Staubli VAL3: editNumField.pgx

public program editNumField(string x_sTitle (dimensions=1), string& x_sItemName[] (dimensions=1), num& x_nItem[] (dimensions=1), num& x_nMin[] (dimensions=1), num& x_nMax[] (dimensions=1))
  local num j
  local num l_nSize
  local num l_nKey
  local string l_sEvent
  local num l_nIndex
  local num l_nField
  local string l_sItem
  local num i
  local string l_sEmpty[2]
  local string l_sString1
  local num l_nFollow
begin
  //  //clear & copy
  //  nView=nFirst=0
  //  call listempty()
  //  call numCopy(x_nItem,nOldValue)
  //  call numCopy(x_nItem,nOffSet)
  //  for j=0 to size(nOffSet)-1
  //    nOffSet[j]=0
  //  endFor
  //  // take the size
  //  l_nSize=size(x_sItemName)-1
  //  // create the LIST
  //  call setSizeList(2,max((6-l_nSize/2)-2,2)-2,20,min((l_nSize+1),12))
  //  call listcreate(x_sTitle)
  //  //
  //  // insert items
  //  //
  //  if nParaAdjustType==1
  //    for j=0 to l_nSize
  //      l_sItem=x_sItemName[j]
  //      if l_sItem!=""
  //        if j==9
  //          call strlength(l_sItem,10)
  //          if x_nItem[j]==0
  //            call listadd(l_sItem+": "+"关")
  //          else
  //            call listadd(l_sItem+": "+"开")
  //          endIf
  //        else
  //          call strlength(l_sItem,10)
  //          call listadd(l_sItem+": "+toString(".3",x_nItem[j]))
  //        endIf
  //        nOffSet[j]=nOffSet[max(j-1,0)]
  //      else
  //        nOffSet[j]=nOffSet[max(j-1,0)]+1
  //      endIf
  //    endFor
  //  endIf
  //  if nParaAdjustType==2
  //    for j=0 to l_nSize
  //      l_sItem=x_sItemName[j]
  //      if l_sItem!=""
  //        if j==7
  //          call strlength(l_sItem,10)
  //          if x_nItem[j]==0
  //            call listadd(l_sItem+": "+"关")
  //          else
  //            call listadd(l_sItem+": "+"开")
  //          endIf
  //        else
  //          call strlength(l_sItem,10)
  //          call listadd(l_sItem+": "+toString(".3",x_nItem[j]))
  //        endIf
  //        nOffSet[j]=nOffSet[max(j-1,0)]
  //      else
  //        nOffSet[j]=nOffSet[max(j-1,0)]+1
  //      endIf
  //    endFor
  //  endIf
  //  if nParaAdjustType==3
  //    for j=0 to l_nSize
  //      l_sItem=x_sItemName[j]
  //      if l_sItem!=""
  //        call strlength(l_sItem,10)
  //        call listadd(l_sItem+": "+toString(".3",x_nItem[j]))
  //        nOffSet[j]=nOffSet[max(j-1,0)]
  //      else
  //        nOffSet[j]=nOffSet[max(j-1,0)]+1
  //      endIf
  //    endFor
  //  endIf
  //  // update the list
  //  call listupdate(0)
  //  do
  //    call clear(0,13)
  //    call typeMenu(8,"OK")
  //    l_nKey=get()
  //    call listevent(l_nKey,l_nIndex,l_sEvent)
  //    // use the offset
  //    i=l_nIndex+nOffSet[max(l_nIndex,0)]
  //    // on Enter Key
  //    if nParaAdjustType==1
  //      if l_nKey==270
  //        if l_nIndex==9
  //          call listcursor(l_nIndex,false)
  //          if size(x_nMin)==size(x_nItem)
  //            // use min and max
  //            l_sEmpty[0]="关"
  //            l_sEmpty[1]="开"
  //            call changeValue(x_nItem[l_nIndex],x_nMin[l_nIndex],x_nMax[l_nIndex],15,nView+nTopY+1,l_sEmpty)
  //          else
  //            l_sEmpty[0]="关"
  //            l_sEmpty[1]="开"
  //            call changeValue(x_nItem[l_nIndex],x_nMin[l_nIndex],x_nMax[l_nIndex],15,nView+nTopY+1,l_sEmpty)
  //          endIf
  //          // UPDATE
  //          call listdel(l_nIndex)
  //          l_sItem=x_sItemName[l_nIndex]
  //          call strlength(l_sItem,10)
  //          call listins(l_sItem+": "+l_sEmpty[x_nItem[l_nIndex]],l_nIndex)
  //          call listupdate(l_nIndex-nView)
  //        else
  //          call listcursor(l_nIndex,false)
  //          if size(x_nMin)==size(x_nItem)
  //            // use min and max
  //            l_sEmpty[0]=""
  //            l_sEmpty[1]=""
  //            call changeValue(x_nItem[i],x_nMin[i],x_nMax[i],15,nView+nTopY+1,l_sEmpty)
  //          else
  //            call changeValue(x_nItem[i],x_nMin,x_nMax,15,nView+nTopY+1,l_sEmpty)
  //          endIf
  //          // UPDATE
  //          call listdel(l_nIndex)
  //          l_sItem=x_sItemName[i]
  //          call strlength(l_sItem,10)
  //          call listins(l_sItem+": "+toString(".3",x_nItem[i]),l_nIndex)
  //          call listupdate(l_nIndex-nView)
  //        endIf
  //      endIf
  //    endIf
  //    if nParaAdjustType==2
  //      if l_nKey==270
  //        if l_nIndex==7
  //          call listcursor(l_nIndex,false)
  //          if size(x_nMin)==size(x_nItem)
  //            // use min and max
  //            l_sEmpty[0]="关"
  //            l_sEmpty[1]="开"
  //            call changeValue(x_nItem[l_nIndex],x_nMin[l_nIndex],x_nMax[l_nIndex],15,nView+nTopY+1,l_sEmpty)
  //          else
  //            l_sEmpty[0]="关"
  //            l_sEmpty[1]="开"
  //            call changeValue(x_nItem[l_nIndex],x_nMin[l_nIndex],x_nMax[l_nIndex],15,nView+nTopY+1,l_sEmpty)
  //          endIf
  //          //UPDATE
  //          call listdel(l_nIndex)
  //          l_sItem=x_sItemName[l_nIndex]
  //          call strlength(l_sItem,10)
  //          call listins(l_sItem+": "+l_sEmpty[x_nItem[l_nIndex]],l_nIndex)
  //          call listupdate(l_nIndex-nView)
  //        else
  //          call listcursor(l_nIndex,false)
  //          if size(x_nMin)==size(x_nItem)
  //            // use min and max
  //            l_sEmpty[0]=""
  //            l_sEmpty[1]=""
  //            call changeValue(x_nItem[i],x_nMin[i],x_nMax[i],15,nView+nTopY+1,l_sEmpty)
  //          else
  //            call changeValue(x_nItem[i],x_nMin,x_nMax,15,nView+nTopY+1,l_sEmpty)
  //          endIf
  //          // UPDATE
  //          call listdel(l_nIndex)
  //          l_sItem=x_sItemName[i]
  //          call strlength(l_sItem,10)
  //          call listins(l_sItem+": "+toString(".3",x_nItem[i]),l_nIndex)
  //          call listupdate(l_nIndex-nView)
  //        endIf
  //      endIf
  //    endIf
  //    if nParaAdjustType==3
  //      if l_nKey==270
  //        //      if l_nIndex==7
  //        //        call listcursor(l_nIndex,false)
  //        //        if size(x_nMin)==size(x_nItem)
  //        //          // use min and max
  //        //          l_sEmpty[0]="关"
  //        //          l_sEmpty[1]="开"
  //        //          call changeValue(x_nItem[l_nIndex],x_nMin[l_nIndex],x_nMax[l_nIndex],15,nView+nTopY+1,l_sEmpty)
  //        //        else
  //        //          l_sEmpty[0]="关"
  //        //          l_sEmpty[1]="开"
  //        //          call changeValue(x_nItem[l_nIndex],x_nMin[l_nIndex],x_nMax[l_nIndex],15,nView+nTopY+1,l_sEmpty)
  //        //        endIf
  //        //        //UPDATE
  //        //        call listdel(l_nIndex)
  //        //        l_sItem=x_sItemName[l_nIndex]
  //        //        call strlength(l_sItem,10)
  //        //        call listins(l_sItem+": "+l_sEmpty[x_nItem[l_nIndex]],l_nIndex)
  //        //        call listupdate(l_nIndex-nView)
  //        //      else
  //        call listcursor(l_nIndex,false)
  //        if size(x_nMin)==size(x_nItem)
  //          // use min and max
  //          l_sEmpty[0]=""
  //          l_sEmpty[1]=""
  //          call changeValue(x_nItem[i],x_nMin[i],x_nMax[i],15,nView+nTopY+1,l_sEmpty)
  //        else
  //          call changeValue(x_nItem[i],x_nMin,x_nMax,15,nView+nTopY+1,l_sEmpty)
  //        endIf
  //        // UPDATE
  //        call listdel(l_nIndex)
  //        l_sItem=x_sItemName[i]
  //        call strlength(l_sItem,10)
  //        call listins(l_sItem+": "+toString(".3",x_nItem[i]),l_nIndex)
  //        call listupdate(l_nIndex-nView)
  //        //      endIf
  //      endIf
  //    endIf
  //    delay(0)
  //  until l_nKey==278 or l_nKey==255
  //  // escape use????
  //  if l_nKey==255
  //    bUseEscape=true
  //    call numCopy(nOldValue,x_nItem)
  //  else
  //    bUseEscape=false
  //  endIf
  //  // exit
  //  call nullKey(l_nKey)
end
